FUNCTION_BLOCK T_AssertionMessageList IMPLEMENTS I_AssertionMessageList
VAR
    _Messages : ARRAY[0..MAX_ASSERTION_MESSAGES] OF T_MaxString;
    _Count : INT;
END_VAR

METHOD AddMessage : BOOL
VAR_INPUT
    Message : T_MaxString;
END_VAR
IF _Count <= MAX_ASSERTION_MESSAGES THEN
    _Messages[_Count] := Message;
    _Count := _Count + 1;
    AddMessage := TRUE;
END_IF
END_METHOD

METHOD Clear
VAR_INPUT
END_VAR
MEMSET(
    destAddr := ADR(_Messages), 
    fillByte := 0, 
    n        := SIZEOF(_Messages));
_Count := 0;
END_METHOD

END_FUNCTION_BLOCK

(* stored: Version 1.1.0.1, ProductVersion 3.1.4024.4
   POU T_AssertionMessageList: Id {e7d5340d-c089-4dbb-ae44-9c00444fa0e8}, SpecialFunc None
   Method AddMessage: Id {41dc59db-d4bf-41a1-b4a5-2d7f6c4a7161}
   Method Clear: Id {81a3ce51-6363-4c36-9872-c4b7a11d1f4c} *)
